PROGRAM INTERNAL PRG_TEST_GLOBAL // A place to call global function blocks (singletons) that can be used by all tests

Sys_Variables.fbSystemVariables();
GVL_Utilities.fbFaultHandler();

END_PROGRAM

(* stored: Version 1.1.0.1, ProductVersion 3.1.4024.11
   POU PRG_TEST_GLOBAL: Id {b2369d3f-a6c6-470b-8f0b-26f76585cbd1}, SpecialFunc None *)
